TYPE "PLCtoMES_MainCheckIn_ext"
VERSION : 0.1
   STRUCT
      Load_Station1ChickInReq : Bool;
      Load_Station2ChickInReq : Bool;
      Load_Station3ChickInReq : Bool;
      Load_Station4ChickInReq : Bool;
      Load_Station5ChickInReq : Bool;
      Load_Station6ChickInReq : Bool;
      Load_Station7ChickInReq : Bool;
      Load_Station8ChickInReq : Bool;
   END_STRUCT;

END_TYPE

